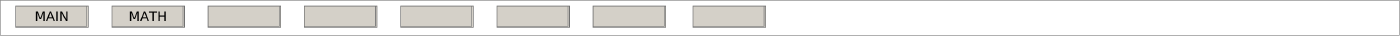
VISUALIZATION Footer  // 1920x50
    Button (21,8 100x30), "MAIN"
        OnMouseClick: change screen: Visualization
    Button (153,8 100x30), "MATH"
    Button (285,8 100x30)
    Button (417,8 100x30)
    Button (549,8 100x30)
    Button (681,8 100x30)
    Button (813,8 100x30)
    Button (950,8 100x30)
END_VISUALIZATION

(* stored: Version 1.1.0.1, ProductVersion 3.1.4024.12
   Visu Footer: Id {3d6eaa1f-e3bc-4cf7-9ac5-cf81c9752ab3} *)
